PROGRAM MAIN
VAR
	stAmsNetId	AT %I*	              : AMSNETID;
	nPort	AT %I*                    : WORD;
	nMasterAxisPosition AT %I*        : DINT;
	nAdditivePositionSetpoiunt AT %Q* : DINT;
	nAdditiveTorqueSetpoint    AT %Q* : INT;   // Unit 0.1%  (10=1%)
	dLatchedPosition AT %I*           : DINT;
	iBrakeSpRaw AT %Q*                : INT := 0;
	//iRotMotorTempRaw AT %I*           : INT := 0;
    fbTemp                            : EL3214;
	bBrakeFreewheelOn AT %Q*          : BOOL;
	bBrakeLockedOn AT %Q*             : BOOL;
    inputDummy AT %I*                 : BOOL;
	inputDigSens1 AT %I*              : BOOL;
	inputDigSens2 AT %I*              : BOOL;
	fbBrakeTorque                     : FB_BrakeTorque;  // Control brake
	fbModePhase                       : FB_ModePhasing;	 // Phasing Mode
	fbRampVelo                        : FB_RampVelo;
	fbModeVelo                        : FB_ModeVelo;     // Velocity Mode
	fbModePos                         : FB_ModePos;      // Positioning Mode
	fbModeHome                        : FB_ModeHome;     // Homing Mode
	fbIndraDrive                      : fbIndraDrive;    // Control of drive
	stStatEpics                       : ST_STAT_EPICS;   // Status to EPICS
	stCmdEpics                        : ST_CMD_EPICS;    // Control to EPICS 
	stCommands                        : ST_AXIS_COMMAND; // Control to drive
	stStatus                          : ST_AXIS_STATUS;  // Status from drive
	eTargetStateOld                   : TARGET_STATE_MACHINE;
	addStartupTorqueTrigger           : BOOL:=FALSE;
	iTorqueCommandValue  AT %Q*       : INT := 0;
END_VAR

// Monitor temperature
ACT_Temperature();
// Control brake
ACT_Brake();


// Enable Axis independent of state
stCommands.bEnableAxis :=stCmdEpics.bEnable;
stCommands.bHaltAxis:=stCmdEpics.bExecute;
stStatEpics.bEnabled:=stStatus.bAxisEnabled;
stCommands.bCmd_ErrorReset:=stCmdEpics.bReset;

IF NOT stCmdEpics.bEnable THEN
  stCmdEpics.bExecute:=FALSE;
END_IF

stCommands.fCommandAcceleration:=GVL_Parameters.fAccDefault;
stCommands.fCommandDeceleration:=GVL_Parameters.fAccDefault;
stCommands.bCmd_DriveControlledHoming:=FALSE;

// Only allow state change if execute is low
IF stCmdEpics.eTargetStateCmd <> stStatEpics.eTargetState AND NOT stCmdEpics.bexecute THEN
	stStatEpics.eTargetState:=stCmdEpics.eTargetStateCmd;
END_IF

//nAdditiveTorqueSetpoint:=0;
//IF NOT  stCmdEpics.bExecute THEN
//	addStartupTorqueTrigger:=TRUE;
//END_IF

CASE stStatEpics.eTargetState OF 
	TARGET_STATE_MACHINE.CONSTANT_VELOCITY:
		fbModeVelo(
            bExecute:=         stCmdEpics.bExecute,
            bReset:=           stCmdEpics.bReset,
			fVelSet:=          stCmdEpics.fVelSet,
			stStatus:=	       stStatus,	
			stCommands:=       stCommands);
			
			//ramp velocity with selected acceleration
			fbRampVelo(bExecute:=stCmdEpics.bExecute,
              fVelSetIn:=fbModeVelo.fSpeedSetpoint,
              iBlockSampleTimeMicroS:=GVL_Parameters.nTaskSampleTime*1000,
              fVelSetOut:=stCommands.fVelocityCommandValue,
              fVelActIn:=stStatus.fActualVelocity/10);
			  
// add extra torque att startup TEST
		//	IF stStatus.bAxisEnabled AND stCmdEpics.bExecute AND stCmdEpics.fVelSet > 0 THEN
		//		IF stStatus.fActualVelocity/10< stCmdEpics.fVelSet/2 THEN
		//	        nAdditiveTorqueSetpoint:=100;  //Add 10% when under x rpm
		//		ELSIF stStatus.fActualVelocity/10 > stCmdEpics.fVelSet/2 THEN
		//			nAdditiveTorqueSetpoint:=40;
		//		END_IF
		//	END_IF

			
	TARGET_STATE_MACHINE.POSITIONING:
		fbModePos(
            bExecute:=         stCmdEpics.bExecute,
            bReset:=           stCmdEpics.bReset,
			fVelSet:=          stCmdEpics.fVelSet,
			fPosSet:=          stCmdEpics.fPosSet,
			stStatus:=         stStatus,	
			stCommands:=       stCommands);
		
	TARGET_STATE_MACHINE.PHASING:
   		fbModePhase(
			bExecute:=         stCmdEpics.bExecute,
            bReset:=           stCmdEpics.bReset,
			stStatus:=	       stStatus,
			dLatchedPosition:= dLatchedPosition,
			ePhaseType:=stCmdEpics.ePhaseCntrlAlg,
			stCommands:=       stCommands);
			
			//ramp velocity with selected acceleration (as long as not phasing)
			IF NOT fbModePhase.bPhasing THEN
              fbRampVelo(bExecute:=stCmdEpics.bExecute,
                fVelSetIn:=fbModePhase.fSpeedSetpoint,
                iBlockSampleTimeMicroS:=GVL_Parameters.nTaskSampleTime*1000,
                fVelSetOut:=stCommands.fVelocityCommandValue,
                fVelActIn:=fbModePhase.fLastSectorVelocity);
			ELSE // if phasing then take setpoint direct from fbModePhase
			  stCommands.fVelocityCommandValue:=fbModePhase.fSpeedSetpoint;
            END_IF
						
	TARGET_STATE_MACHINE.HOMING:
        fbModeHome( 
            bExecute:=         stCmdEpics.bExecute,
            bReset:=           stCmdEpics.bReset,
			fVelSet:=          stCmdEpics.fVelSet,
			fPosSet:=          stCmdEpics.fPosSet,
			stStatus:=	       stStatus,	
			stCommands:=       stCommands);
			
	TARGET_STATE_MACHINE.TORQUE:
		stCommands.eOperationMode:=E_OPERATION_MODE_NO.eSecondaryOpMode7;
	    stCommands.eMotionMode :=e_Motion_mode.eJogPositive;
	
	  ELSE  // No valid state
		  
		stCmdEpics.bExecute:=FALSE;
        stCmdEpics.bEnable:=FALSE;
		stCommands.fVelocityCommandValue:=0;
		stCommands.fCommandVelocity:=0;
		
END_CASE

IF NOT stCmdEpics.bExecute THEN
	stCommands.fVelocityCommandValue:=0;
END_IF

// TODO: Why I put this here?
stCommands.eMotionMode:=E_MOTION_MODE.eStop;

// Rexroth FB
fbIndraDrive(
	AmsNetId:= stAmsNetId, 
	AdsAddr_Port:= nPort, 
	stAxisCommands:= stCommands, 
	stDriveStatus:= , 
	stAxisStatus=> stStatus, 
	stDriveCommands=> );

// Calculate values for status in EPICS
stStatEpics.fSetVelRaw:= DINT_TO_LREAL(MAIN.fbIndraDrive.stDriveCommands.nS40_VelocityCommandValue)/10000;	
stStatEpics.fActPos:=stStatus.fActualPosition;
stStatEpics.fActTorque:=stStatus.fActualTorque;
stStatEpics.fActVel:=stStatus.fActualVelocity/10;

// Error handling
ACT_Error();

eTargetStateOld:=stStatEpics.eTargetState;

ACTION ACT_Brake:
// Function: Control of brake for simulation of traction
// Use at target test rig
// Author: Anders Sandström 2019

bBrakeFreewheelOn:=stCmdEpics.bFreeWheelOnOnCmd;
bBrakeLockedOn:=stCmdEpics.bBrakeLockOnCmd;

fbBrakeTorque(iTorqueValueinNm:=stCmdEpics.fBrakeSpNm);
iBrakeSpRaw:=fbBrakeTorque.iTorqueScaled;
END_ACTION

ACTION ACT_Diag:
// Function: Some parameters just for debugging
// Note: Do not need to be executed, can be watched online anyway..
// Author: Anders Sandström 2019

	stCommands.bCmd_ActivateParameterMode;//True puts the drive in parameter mode
	stCommands.bCmd_DisableLimits;// True disables monitoring of errors
	stCommands.bCmd_DriveControlledHoming;// True starts homing procedure defined in the drive
	stCommands.bCmd_ErrorReset;
	stCommands.bCmd_ExitParameterMode;
	stCommands.bCmd_RunVirtualMater;// Jog command to the virtual master
	stCommands.bCmd_SetAbsolutePosition;
	stCommands.bCommandPositionChange;// Drive moves to the current target position, when bCommandVAlueAccept toggled, drive moves to the new target position
	stCommands.bCommandValueAccept;// Used in "Drive positioning Mode" to update the target position when toggled
	stCommands.bEnableAxis;
	stCommands.bHaltAxis;// Performs halt on the drive, bEnableaxis has to be TRUE
	stCommands.bPositionCommandValue;//0=Absolute;1=Relative
	stCommands.eMotionMode;
	stCommands.eOperationMode;
	stCommands.fCommandAcceleration;// Acceleration used for positioning and jogging
	stCommands.fCommandDeceleration;// Deceleration used for positioning and jogging
	stCommands.fCommandPosition;
	stCommands.fCommandVelocity;// Velocity used for positioning and jogging
	stCommands.fFeedrateOverride;// Parameter used for adjustment of the velocity (0,100)%
	stCommands.fTorqueLimit;
	stCommands.fVelocityCommandValue;// S40, velocity used for positining and jogging (in velocity mode)
	stStatus.bAxisEnabled;
END_ACTION

ACTION ACT_Error:
// Function: Error handling
// Author: Anders Sandström 2019

IF stStatEpics.eTargetState = TARGET_STATE_MACHINE.PHASING THEN
  IF fbModePhase.bError AND NOT stStatEpics.bError THEN
	  stStatEpics.bError:=fbModePhase.bError;
	  stStatEpics.nErrorId:=fbModePhase.nErrorId;
	  stStatEpics.sErrorStr:=fbModePhase.sErrorStr;
  END_IF
  
ELSIF stStatEpics.eTargetState = TARGET_STATE_MACHINE.CONSTANT_VELOCITY THEN
   IF fbModeVelo.bError AND NOT stStatEpics.bError THEN
	  stStatEpics.bError:=fbModeVelo.bError;
	  stStatEpics.nErrorId:=fbModeVelo.nErrorId;
	  stStatEpics.sErrorStr:=fbModeVelo.sErrorStr;
  END_IF
  
ELSIF stStatEpics.eTargetState = TARGET_STATE_MACHINE.POSITIONING THEN
  IF fbModePos.bError AND NOT stStatEpics.bError THEN
	  stStatEpics.bError:=fbModePos.bError;
	  stStatEpics.nErrorId:=fbModePos.nErrorId;
	  stStatEpics.sErrorStr:=fbModePos.sErrorStr;
  END_IF
  
ELSIF stStatEpics.eTargetState = TARGET_STATE_MACHINE.HOMING THEN
  IF fbModeHome.bError AND NOT stStatEpics.bError THEN
	  stStatEpics.bError:=fbModeHome.bError;
	  stStatEpics.nErrorId:=fbModeHome.nErrorId;
	  stStatEpics.sErrorStr:=fbModeHome.sErrorStr;
  END_IF
  
END_IF


IF stcmdEpics.bReset THEN
	stStatEpics.bError:=FALSE;
	stStatEpics.nErrorId:=GVL_ErrorCodes.nErrorCodeOKId;
	stStatEpics.sErrorStr:=GVL_ErrorCodes.nErrorCodeOKStr;
	stStatEpics.bBrake1TempAlarm:=FALSE;
	stStatEpics.bBrake2TempAlarm:=FALSE;
END_IF
END_ACTION

ACTION ACT_Temperature:
// Function: Monitor tempertures
// Interlock motion on temperatures
// Author: Anders Sandström 2019

fbTemp(En:=TRUE);

IF fbTemp.bError THEN
	stCmdEpics.bExecute:=0;
	stCmdEpics.bEnable:=0;
END_IF

stStatEpics.fActTemp:=fbTemp.iAi_Ch1_Value/10.0;
stStatEpics.fBrakeActTemp1:=fbTemp.iAi_Ch2_Value/10.0;
stStatEpics.fBrakeActTemp2:=fbTemp.iAi_Ch3_Value/10.0;

// Motor Temperature Monitoring Interlock
IF (stStatEpics.fActTemp >= GVL_Parameters.nMaxMotorTemperature)  OR fbTemp.iAi_Ch1_Stat >0 THEN
	stCmdEpics.bEnable:= FALSE;
	stCmdEpics.bExecute:= FALSE;	
END_IF

//Brake temperature monitoring Interlock 1
IF (stStatEpics.fBrakeActTemp1 >= GVL_Parameters.nMaxBrakeTemperature) OR fbTemp.iAi_Ch2_Stat >0 OR stStatEpics.bBrake1TempAlarm THEN
	stCmdEpics.bEnable:= FALSE;
	stCmdEpics.bExecute:= FALSE;		
    stStatEpics.bBrake1TempAlarm:=TRUE; 
END_IF
//Brake temperature monitoring Interlock 2
IF (stStatEpics.fBrakeActTemp2 >= GVL_Parameters.nMaxBrakeTemperature) OR fbTemp.iAi_Ch3_Stat >0 OR stStatEpics.bBrake2TempAlarm THEN
	stCmdEpics.bEnable:= FALSE;
	stCmdEpics.bExecute:= FALSE;		
    stStatEpics.bBrake2TempAlarm:=TRUE; 
END_IF
END_ACTION

END_PROGRAM

(* stored: Version 1.1.0.1, ProductVersion 3.1.4024.0
   POU MAIN: Id {40828a63-f1c1-40a3-a7c5-8a47be350a36}, SpecialFunc None
   Action ACT_Brake: Id {a8ef5cdf-33a2-41f9-b34e-1a95819e04c4}
   Action ACT_Diag: Id {2a0ea7d8-8ff8-4796-ae8a-6c3ebb6f7955}
   Action ACT_Error: Id {6316e704-a716-4c28-824a-a22fe5448145}
   Action ACT_Temperature: Id {ec2bd795-c2d7-49be-acd7-2671eaea481b} *)
